FUNCTION_BLOCK T_RoboConnect_WhenCalled_IsConnectedTrue EXTENDS T_UnitTestBase
VAR
  robot : I_RoboConnect;
  timeOutTimer : TON;
  myTestState, prevState : (INIT, ARRANGE, ACT, ASSERT) := INIT;
  expected, actual : BOOL;
  counter : UINT;
END_VAR

CASE myTestState OF
  INIT:
    StateChanged();
    myTestState := ARRANGE;

  ARRANGE:
    StateChanged();

    expected := TRUE;
    myTestState := ACT;

  ACT:
    robot.Connect();
    myTestState := ASSERT;

  ASSERT:

    IF robot.Connected OR timeOutTimer.Q THEN
      actual := robot.Connected;
      assertion.AssertEquals_BOOL(expected, actual, 'IsConnected := TRUE');
      TestFinished();
      myTestState := INIT;
      // dont disconnect here, connection is required for the next test
    END_IF

END_CASE

timeOutTimer(IN := myTestState = ASSERT);

METHOD FB_init : BOOL
VAR_INPUT
  bInitRetains : BOOL; // if TRUE, the retain variables are initialized (warm start / cold start)
  bInCopyCode : BOOL; // if TRUE, the instance afterwards gets moved into the copy code (online change)
  TestSuite : tcl_SimpleUnitTestLibrary.I_TestSuite;
  robot : I_TcRobot;
  timeout : TIME;
END_VAR
THIS^.robot := robot;
THIS^.timeOutTimer.PT := timeout;
END_METHOD

METHOD PRIVATE StateChanged : BOOL
IF  myTestState = prevState THEN
  RETURN;
END_IF

prevState := myTestState;
StateChanged := TRUE;
END_METHOD

METHOD WaitForCycles : BOOL
VAR_INPUT
  maxCount : UINT;
END_VAR
counter := counter + 1;

IF counter = maxCount THEN
  counter := 0;
  WaitForCycles := TRUE;
END_IF
END_METHOD

END_FUNCTION_BLOCK

(* stored: Version 1.1.0.1
   POU T_RoboConnect_WhenCalled_IsConnectedTrue: Id {244d12de-a76c-4ea5-b81b-43bad9781c8a}, SpecialFunc None
   Method FB_init: Id {13d14303-026c-0553-1a6e-eed98e3e944a}
   Method StateChanged: Id {8273eccb-e48e-40e1-905c-4c159a8023fc}
   Method WaitForCycles: Id {6d391f95-bdfa-4a40-9c7e-b0ac0a32a831} *)
